FUNCTION_BLOCK NationalCylinderControl (* Basic Function Block Type *)
  (* Standard: 61499-2 *)
  (* Version 0.0, 12/9/2021, e_net, nxtControl GmbH, Template *)
  PACKAGE Main;
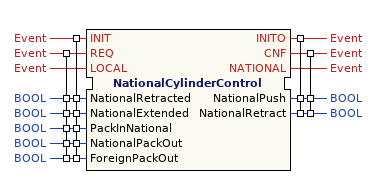
  EVENT_INPUT
    INIT WITH NationalRetracted, NationalExtended, PackInNational, NationalPackOut, ForeignPackOut; (* Initialization Request *)
    REQ WITH NationalRetracted, NationalExtended, PackInNational, NationalPackOut, ForeignPackOut; (* Normal Execution Request *)
    LOCAL;
  END_EVENT
  EVENT_OUTPUT
    INITO WITH NationalPush, NationalRetract; (* Initialization Confirm *)
    CNF WITH NationalPush, NationalRetract; (* Execution Confirmation *)
    NATIONAL;
  END_EVENT
  VAR_INPUT
    NationalRetracted : BOOL;
    NationalExtended : BOOL;
    PackInNational : BOOL;
    NationalPackOut : BOOL;
    ForeignPackOut : BOOL;
  END_VAR
  VAR_OUTPUT
    NationalPush : BOOL;
    NationalRetract : BOOL;
  END_VAR
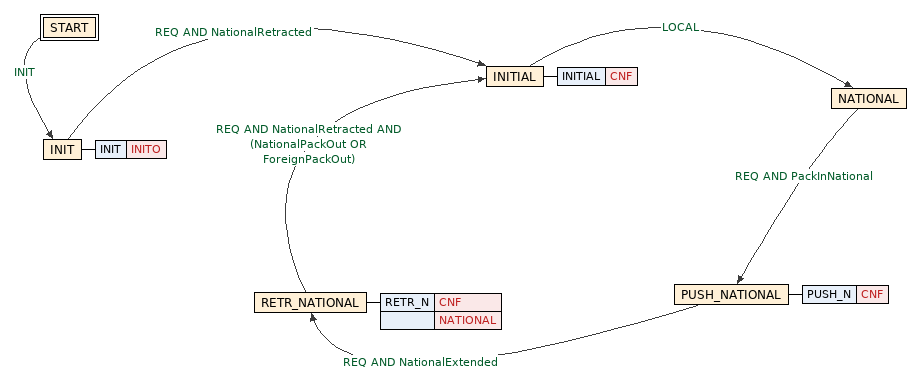
  EC_STATES
    START; (* Initial State *)
    INIT : INIT -> INITO; (* Initialization *)
    INITIAL : INITIAL -> CNF;
    PUSH_NATIONAL : PUSH_N -> CNF;
    RETR_NATIONAL : RETR_N -> CNF, -> NATIONAL;
    NATIONAL;
  END_STATES
  EC_TRANSITIONS
    START TO INIT := INIT;
    INIT TO INITIAL := REQ AND NationalRetracted;
    RETR_NATIONAL TO INITIAL := REQ AND NationalRetracted AND (NationalPackOut OR ForeignPackOut);
    NATIONAL TO PUSH_NATIONAL := REQ AND PackInNational;
    PUSH_NATIONAL TO RETR_NATIONAL := REQ AND NationalExtended;
    INITIAL TO NATIONAL := LOCAL;
  END_TRANSITIONS
  ALGORITHM INIT IN ST: (* Initialization algorithm *)
NationalPush:= FALSE;
NationalRetract:= TRUE;
  END_ALGORITHM
  ALGORITHM INITIAL IN ST:
NationalRetract:=FALSE;
  END_ALGORITHM
  ALGORITHM PUSH_N IN ST:
NationalPush:=TRUE;
  END_ALGORITHM
  ALGORITHM RETR_N IN ST:
NationalPush:=FALSE;
NationalRetract:=TRUE;
  END_ALGORITHM
END_FUNCTION_BLOCK
